TYPE ST_SensorRaw :
    STRUCT
		(* EL3204 - 1*)
        temperatureEvaporatingOut		AT %I*	: INT;  (* Verdampfungstemperatur in °C (Ausgang) *)
        temperatureEvaporatingIn		AT %I*	: INT;  (* Verdampfungstemperatur in °C (Eingang) *)
        temperatureFlow	 				AT %I*	: INT;  (* Vorlauftemperatur in °C *)
        temperatureReturn				AT %I*	: INT;  (* Rücklauftemperatur in °C *)
		
		(* EL3204 - 2*)
        temperatureOverheatedGas		AT %I*	: INT;  (* Saugtemperatur des überhitzten Gases *)
        bufferTopTemperature			AT %I*	: INT;  (* Temperatur des Puffers oben in °C *)
		bufferMiddleTemperature			AT %I*	: INT;  (* Temperatur des Puffers in der Mitte °C *)	
		boilerTemperature				AT %I*	: INT;  (* Boiler-Temperatur oben °C *)	
		
		(* EL3204 - 3*)
		temperatureSourceWaterIn		AT %I*	: INT;  (* Quellwassertemperatur Eingang in °C *)
		temperatureSourceWaterOut		AT %I*	: INT;  (* Quellwassertemperatur Ausgang in °C *)		

		(* EL3122 - 4-20mA*)
        pressureHigh					AT %I*	: INT;  (* Hochdruck Kältekreis in bar *)
        pressureLow						AT %I*	: INT;  (* Niederdruck Kältekreis in bar *)
		
		(* EL3064 - 0-10V* or EL3102 -  +/-10V *)
        pressureDifferenceEvaporator	AT %I*	: INT;  (* Druckdifferenz im Verdampfer in mbar *)
    END_STRUCT
END_TYPE

(* stored: Version 1.1.0.1
   DUT ST_SensorRaw: Id {946a79e1-c3d0-4e8b-887c-36a900db2305} *)
